TYPE ST_TrayPositionConfig :
STRUCT
    fLiftStationX : LREAL;
    fRackStationX : LREAL;
    fStandbyZ : LREAL;
    fPickupLevelZ : LREAL;
    aLayer : ARRAY[1..5] OF ST_TrayLayerPositionConfig;
END_STRUCT
END_TYPE

(* stored: Version 1.1.0.1, ProductVersion 3.1.4026.20
   DUT ST_TrayPositionConfig: Id {261c9dc4-1cf6-4e77-a507-902d0773d91f} *)
